// TwinCAT 3 PLC project PLC1
// ProgramVersion: 3.1.4026.15
// libraries:
//   Tc2_ModbusRTU, * (Beckhoff Automation GmbH)
//   Tc2_ModbusSrv, * (Beckhoff Automation GmbH)
//   Tc2_Standard, * (Beckhoff Automation GmbH)
//   Tc2_System, * (Beckhoff Automation GmbH)
// project tree:
//   GVLs/ FIO.TcGVL, GVL.TcGVL
//   / PlcTask.TcTTO
//   POUs/FactoryIO/ AssignInsOuts.TcPOU
//   POUs/FactoryIO/NOT USED/ FB_FactoryIO_ReadInputs_.TcPOU, FB_FactoryIO_WriteOutputs.TcPOU
//   POUs/ MAIN.TcPOU
//   POUs/SubRoutines/ F_Faults.TcPOU, C_Input_Conveyor.TcPOU, B_Machine_Center.TcPOU, E_Output_Conveyor.TcPOU, D_Stacker_Crane.TcPOU, A_System_Start.TcPOU
// real-time tasks:
//   TASK PlcTask: cycle T#10ms, priority 20, ADS port 350

CONFIGURATION PLC1
    RESOURCE PLC ON TwinCAT3
        TASK PlcTask(INTERVAL := T#10ms, PRIORITY := 20);
        PROGRAM MAIN WITH PlcTask : MAIN;
    END_RESOURCE
END_CONFIGURATION

// ---- GVLs/FIO.TcGVL
{attribute 'qualified_only'}
VAR_GLOBAL
	
//HMI
	



//Factory IO 
	//Inputs
		// MACH CNTR BUSY
			b_IN_0: BOOL;
		// MACH CNTR ERR
			b_IN_1: BOOL;
		// CONTAIN EMIT PE
			b_IN_2: BOOL;
		// BASE VISION SENS
			b_IN_3: BOOL;
		// INPUT CONV 1 PE
			b_IN_4: BOOL;
		// INPUT PICKUP PE
			b_IN_5: BOOL;
		// OUT DEP CONV PE
			b_IN_6: BOOL;
		// OUT CONV 1 PE
			b_IN_7: BOOL;
		// OUT CONV 2 PE
			b_IN_8: BOOL;
		// CRANE MOVE X
			b_IN_9: BOOL;
		// CRANE MOVE Z
			b_IN_10: BOOL;
		// CRANE LEFT LS
			b_IN_11: BOOL;
		// CRANE RIGHT LS
			b_IN_12: BOOL;
		// CRANE MID LS
			b_IN_13: BOOL;
		// UNUSED
			b_IN_14: BOOL;
		// UNUSED
			b_IN_15: BOOL;
		// UNUSED
			b_IN_64: BOOL;
	
	
		// Machining Center  Progress
			r_IN_0: WORD;
		//Light Array Emitter
			r_IN_1: WORD;
//Outputs
		// RAW MAT EMIT
			b_OUT_0: BOOL;
		// MACH LIDS
			b_OUT_1: BOOL;
		// CONTAIN CONV EMIT
			b_OUT_2: BOOL;
		// CONTAIN CONV MS
			b_OUT_3: BOOL := FALSE;
		// CONV PICK MS
			b_OUT_4: BOOL;
		// OUT DEP CONV MS
			b_OUT_5: BOOL;
		// OUT CONV 1 MS
			b_OUT_6: BOOL;
		// OUT CONV 2 MS
			b_OUT_7: BOOL;
		// OUT CONV REMOVE
			b_OUT_8: BOOL;
		// CRANE LIFT
			b_OUT_9: BOOL;
		// CRANE LEFT
			b_OUT_10: BOOL;
		// CRANE RIGHT
			b_OUT_11: BOOL;
		// INPUT CONV 1 MS
			b_OUT_12: BOOL;
		// CNC MACH RESET
			b_OUT_13: BOOL;
		// UNUSED
			b_OUT_14: BOOL;
		// UNUSED
			b_OUT_15: BOOL;
		// UNUSED
			b_OUT_16: BOOL;
		
		
		//Stacker Crane Target Position
			r_out_0: WORD;

END_VAR

// ---- GVLs/GVL.TcGVL
{attribute 'qualified_only'}
VAR_GLOBAL
	bSystemStart : BOOL := FALSE; 			//HMI Start
    bAutoMode : BOOL := FALSE;				//HMI Auto
    bCNCOn : BOOL := FALSE;					//HMI CNC ON
    bRetrieveCMD : BOOL := FALSE;			//HMI Retrieve command
    bReset : BOOL := FALSE;					//HMI Reset

    iProductID : INT := 4000;				//Current Product ID
    arrStoredIDs : ARRAY[1..15] OF INT := [0];		//Array of stored products
    arrExitIDs : ARRAY[1..15] OF INT:= [0];		//Array of exited products
    iStorageCount : INT := 0;				//num of stored items
    iExitCount : INT := 0;					//num of retrieved items

    bFaultDetected : BOOL := FALSE;			//global fault indicator
    sFaultMessage : STRING := '';			//global fault message
	
	// Indicates System is in run state
	SystemRun: BOOL := FALSE;
	// Box ID of queued Container
	QueuedBoxID: INT := 0;
	// Box Waiting for crane
	ContainerWaitingInput: BOOL := FALSE;
	
	ContainerWaitingOutput : BOOL := FALSE;
	
	//Warehouse has reached 15 box capacity
	WarehouseFull : BOOL := FALSE;
	
	//If crane is in input mode
	InputtingBoxes : BOOL := TRUE;
	//If crane is in output mode
	OutputtingBoxes : BOOL := FALSE;
	//Commanded location of crane
	CommandedLocation : INT :=1;
END_VAR

// ---- POUs/MAIN.TcPOU
PROGRAM MAIN
VAR
END_VAR

AssignInsOuts();


A_System_Start();
IF gvl.bSystemStart THEN
	IF GVL.SystemRun THEN
		B_Machine_Center();
		C_Input_Conveyor();
		D_Stacker_Crane();
		E_Output_Conveyor();
	END_IF
    F_Faults();
END_IF

END_PROGRAM

// ---- POUs/FactoryIO/AssignInsOuts.TcPOU
PROGRAM AssignInsOuts
VAR
	//Factory IO
	FactoryIO_Ins : ARRAY [0..15] OF BYTE;
	FactoryIO_RegIns : ARRAY [0..7] OF WORD;
	FactoryIO_Outs : ARRAY [0..15] OF BYTE;
	FactoryIO_RegOuts : ARRAY [0..7] OF WORD;
	
	//FIO Function Blocks
	FactoryIO_ReadInsFB : FB_MBReadInputs;
	FactoryIO_WriteOutsFB : FB_MBWriteCoils;
	FactoryIO_ReadRegsFB : FB_MBReadInputRegs;
	FactoryIO_WriteRegsFB : FB_MBWriteRegs;
	
END_VAR

//Reads Inputs and Writes Outputs to FactoryIO


FactoryIO_ReadInsFB(
	sIPAddr:= '127.0.0.1' , 
	nTCPPort:= 505, 
	nUnitID:= 1, 
	nQuantity:= 16, 
	nMBAddr:= 0, 
	cbLength:= SIZEOF(AssignInsOuts.FactoryIO_Ins), 
	pDestAddr:= ADR(AssignInsOuts.FactoryIO_Ins), 
	bExecute:= TRUE, 
	tTimeout:= T#1S, 
	bBusy=> , 
	bError=> , 
	nErrId=> , 
	cbRead=> );
FactoryIO_ReadInsFB(bExecute:=FALSE);


FactoryIO_ReadRegsFB(
	sIPAddr:= '127.0.0.1', 
	nTCPPort:= 505, 
	nUnitID:= 1, 
	nQuantity:= 8, 
	nMBAddr:= 0, 
	cbLength:=  SIZEOF(AssignInsOuts.FactoryIO_RegIns), 
	pDestAddr:= ADR(AssignInsOuts.FactoryIO_RegIns), 
	bExecute:= TRUE, 
	tTimeout:= T#1S, 
	bBusy=> , 
	bError=> , 
	nErrId=> , 
	cbRead=> );
FactoryIO_ReadRegsFB(bExecute := FALSE);



FactoryIO_WriteOutsFB(
	sIPAddr:= '127.0.0.1', 
	nTCPPort:= 505, 
	nUnitID:= 1, 
	nQuantity:= 16, 
	nMBAddr:= 0, 
	cbLength:= SIZEOF(AssignInsOuts.FactoryIO_Outs), 
	pSrcAddr:= ADR(AssignInsOuts.FactoryIO_Outs), 
	bExecute:= TRUE, 
	tTimeout:= T#1S, 
	bBusy=> , 
	bError=> , 
	nErrId=> );
FactoryIO_WriteOutsFB(bExecute:=FALSE);



FactoryIO_WriteRegsFB(
	sIPAddr:= '127.0.0.1', 
	nTCPPort:= 505, 
	nUnitID:= 1, 
	nQuantity:= 8, 
	nMBAddr:= 0, 
	cbLength:= SIZEOF(AssignInsOuts.FactoryIO_regOuts), 
	pSrcAddr:= ADR(AssignInsOuts.FactoryIO_regOuts), 
	bExecute:= TRUE, 
	tTimeout:= T#1S, 
	bBusy=> , 
	bError=> , 
	nErrId=> );
FactoryIO_WriteRegsFB(bExecute := FALSE);
	




//Link Inputs from FactoryIO
FIO.b_IN_0 :=  FactoryIO_Ins [0].0;
FIO.b_IN_1 :=  FactoryIO_Ins [0].1;
FIO.b_IN_2 :=  FactoryIO_Ins [0].2;
FIO.b_IN_3 :=  FactoryIO_Ins [0].3;
FIO.b_IN_4 :=  FactoryIO_Ins [0].4;
FIO.b_IN_5 :=  FactoryIO_Ins [0].5;
FIO.b_IN_6 :=  FactoryIO_Ins [0].6;
FIO.b_IN_7 :=  FactoryIO_Ins [0].7;
FIO.b_IN_8 :=  FactoryIO_Ins [1].0;
FIO.b_IN_9 :=  FactoryIO_Ins [1].1;
FIO.b_IN_10 :=  FactoryIO_Ins [1].2;
FIO.b_IN_11 :=  FactoryIO_Ins [1].3;
FIO.b_IN_12 :=  FactoryIO_Ins [1].4;
FIO.b_IN_13 :=  FactoryIO_Ins [1].5;
FIO.b_IN_14 :=  FactoryIO_Ins [1].6;
FIO.b_IN_15 :=  FactoryIO_Ins [1].6;

FIO.r_IN_0 := FactoryIO_RegIns [0];
FIO.r_IN_1 := FactoryIO_RegIns [1];


//Link Outputs to FactoryIO
FactoryIO_Outs [0].0 := FIO.b_OUT_0;
FactoryIO_Outs [0].1 := FIO.b_OUT_1;
FactoryIO_Outs [0].2 := FIO.b_OUT_2;
FactoryIO_Outs [0].3 := FIO.b_OUT_3;
FactoryIO_Outs [0].4 := FIO.b_OUT_4;
FactoryIO_Outs [0].5 := FIO.b_OUT_5;
FactoryIO_Outs [0].6 := FIO.b_OUT_6;
FactoryIO_Outs [0].7 := FIO.b_OUT_7;
FactoryIO_Outs [1].0 := FIO.b_OUT_8;
FactoryIO_Outs [1].1 := FIO.b_OUT_9;
FactoryIO_Outs [1].2 := FIO.b_OUT_10;
FactoryIO_Outs [1].3 := FIO.b_OUT_11;
FactoryIO_Outs [1].4 := FIO.b_OUT_12;
FactoryIO_Outs [1].5 := FIO.b_OUT_13;

FactoryIO_RegOuts[0] := FIO.r_out_0;

END_PROGRAM

// ---- POUs/SubRoutines/A_System_Start.TcPOU
PROGRAM A_System_Start
VAR

	INITIALIZED: BOOL;
	i: INT;
END_VAR




IF GVL.bSystemStart AND NOT GVL.SystemRun AND NOT INITIALIZED THEN	
	INITIALIZED := TRUE;
	GVL.SystemRun := TRUE;
	FIO.b_OUT_2 := TRUE;//Starts Emitter
	FIO.b_OUT_3 := FALSE;// Stops conveyor 1
	FIO.b_OUT_12 := FALSE;// Stops Conveyor 2
	FIO.b_OUT_4 := FALSE;// Stops Conveyor 3
	gvl.iProductID := 4000;
	GVL.QueuedBoxID := 0;
	
	FOR i := 0 TO 15 DO
		GVL.arrStoredIDs[i] := 0;
		GVL.arrExitIDs[i] := 0;
	END_FOR;
	gvl.CommandedLocation := 1;
	gvl.InputtingBoxes := TRUE;
	GVL.OutputtingBoxes := FALSE;
END_IF

GVL.SystemRun := GVL.bSystemStart;

IF GVL.bReset THEN
	GVL.SystemRun := FALSE;
	INITIALIZED := FALSE;
END_IF

END_PROGRAM

// ---- POUs/SubRoutines/B_Machine_Center.TcPOU
PROGRAM B_Machine_Center
VAR

END_VAR

FIO.b_OUT_1 := FALSE;
FIO.b_OUT_0 := FALSE; //Sets raw emitter to default off
IF (NOT FIO.b_IN_0) AND FIO.b_IN_2  THEN
	FIO.b_OUT_0 := TRUE;
	FIO.b_OUT_1 := TRUE;
	
END_IF

END_PROGRAM

// ---- POUs/SubRoutines/C_Input_Conveyor.TcPOU
PROGRAM C_Input_Conveyor
VAR


END_VAR


// When no containers queued for crane.
IF NOT GVL.ContainerWaitingInput THEN 
	//If there is a full container, move it along the conveyor
	IF FIO.b_IN_2 AND FIO.b_IN_3 THEN
		FIO.b_OUT_2 := FALSE;//Stops Emitter
		FIO.b_OUT_3 := TRUE;// Starts Conveyor 1
		FIO.b_OUT_12 := TRUE;// Starts Conveyor 2
	END_IF
	
	//If the conveyor reaches the first sensor, it stops the first section of the conveyor, starts the third, and emits a new empty container
	IF  FIO.b_IN_4 THEN
		FIO.b_OUT_2 := TRUE; // Emit new container
		FIO.b_OUT_3 := FALSE;// Stops conveyor 1
		FIO.b_OUT_12 := TRUE;// Starts Conveyor 2
		FIO.b_OUT_4 := TRUE;// Starts Conveyor 3
	END_IF
	//If the crane has a container in its loading queue, it stops the conveyor until it is picked up.
	IF  FIO.b_IN_5 THEN
		FIO.b_OUT_2 := FALSE;//Stops emitter
		//GVL.QueuedBoxID := GVL.iProductID;
		//GVL.iProductID := GVL.iProductID +1;
		GVL.ContainerWaitingInput := TRUE;//Sets box waiting to true
		FIO.b_OUT_12 := FALSE;	// stops conveyor 2
		FIO.b_OUT_4 := FALSE;	//stops conveyor 3
	END_IF
END_IF

// If one container is queued for crane
IF GVL.ContainerWaitingInput THEN 
	//If there is a full container, move it along the conveyor
	IF FIO.b_IN_2 AND FIO.b_IN_3 THEN
		FIO.b_OUT_3 := TRUE;// Starts Conveyor 1
		FIO.b_OUT_12 := TRUE;// Starts Conveyor 2
	END_IF
	
	//If the conveyor reaches the first sensor, it stops both sections of the conveyor
	IF  FIO.b_IN_4 THEN
		FIO.b_OUT_3 := FALSE;// Stops conveyor 1
		FIO.b_OUT_12 := FALSE;// Stops Conveyor 2
	END_IF
	
	//If the crane has a container in its loading queue, it stops the conveyor until it is picked up.
	IF  NOT FIO.b_IN_5 THEN
		GVL.ContainerWaitingInput := FALSE;//Sets container waiting to false. Switches to first statement
	END_IF
END_IF

END_PROGRAM

// ---- POUs/SubRoutines/D_Stacker_Crane.TcPOU
PROGRAM D_Stacker_Crane
VAR

	// Current Crane position state
	CranePosition: INT := 0;
	timer : TON;

END_VAR




IF gvl.InputtingBoxes AND (NOT GVL.OutputtingBoxes) THEN
	CASE CranePosition OF
	0://Waiting for command
		FIO.r_out_0:= 99; 		// Crane Position
		FIO.b_OUT_9 := FALSE; 	// Crane Lift
		FIO.b_OUT_10 := FALSE;	//Crane Left (DROPOFF)
		FIO.b_OUT_11 := FALSE;	//Crane Right (Receive)
		timer(IN:= TRUE, PT:= T#500MS, Q=> , ET=> );
		IF GVL.ContainerWaitingInput AND timer.q THEN
			CranePosition := 1;
			timer(IN := FALSE);
		END_IF
	1://Default Position lowered
		FIO.r_out_0:= 99; 		// Crane Position
		FIO.b_OUT_9 := FALSE; 	// Crane Lift
		FIO.b_OUT_10 := FALSE;	//Crane Left (DROPOFF)
		FIO.b_OUT_11 := FALSE;	//Crane Right (Receive)
		timer(IN:= TRUE, PT:= T#500MS, Q=> , ET=> );
		IF (NOT (FIO.b_IN_9 OR FIO.b_IN_10)) AND FIO.b_IN_13 AND timer.q THEN
			CranePosition := 10;
			timer(IN := FALSE);
		END_IF
	10://Pickup lowered
		FIO.r_out_0:= 99; 		// Crane Position
		FIO.b_OUT_9 := FALSE; 	// Crane Lift
		FIO.b_OUT_10 := FALSE;	//Crane Left (DROPOFF)
		FIO.b_OUT_11 := TRUE;	//Crane Right (Receive)
		timer(IN:= TRUE, PT:= T#500MS, Q=> , ET=> );
		IF (NOT (FIO.b_IN_9 OR FIO.b_IN_10)) AND FIO.b_IN_12 AND timer.q THEN
			CranePosition := 20;
			timer(IN := FALSE);
		END_IF
	20://Pickup raised
		FIO.r_out_0:= 99; 		// Crane Position
		FIO.b_OUT_9 := TRUE; 	// Crane Lift
		FIO.b_OUT_10 := FALSE;	//Crane Left (DROPOFF)
		FIO.b_OUT_11 := TRUE;	//Crane Right (Receive)
		timer(IN:= TRUE, PT:= T#500MS, Q=> , ET=> );
		IF timer.Q  THEN
			CranePosition := 30;
			timer(IN := FALSE);
		END_IF
	30://DefaultPosition raised
		FIO.r_out_0:= 99; 		// Crane Position
		FIO.b_OUT_9 := TRUE; 	// Crane Lift
		FIO.b_OUT_10 := FALSE;	//Crane Left (DROPOFF)
		FIO.b_OUT_11 := FALSE;	//Crane Right (Receive)
		IF (NOT (FIO.b_IN_9 OR FIO.b_IN_10)) AND FIO.b_IN_13  THEN
			CranePosition := 40;
		END_IF
	40://Commanded Location queue lowered
		FIO.r_out_0:= TO_WORD(gvl.CommandedLocation); 		// Crane Position
		FIO.b_OUT_9 := FALSE; 	// Crane Lift
		FIO.b_OUT_10 := FALSE;	//Crane Left (DROPOFF)
		FIO.b_OUT_11 := FALSE;	//Crane Right (Receive)
		timer(IN:= TRUE, PT:= T#500MS, Q=> , ET=> );
		IF (NOT FIO.b_IN_9) AND (NOT FIO.b_IN_10) AND FIO.b_IN_13 AND timer.q THEN
			CranePosition := 50;
			timer(IN := FALSE);
		END_IF
	50://Commanded Location queue raised
		FIO.r_out_0:= TO_WORD(gvl.CommandedLocation); 		// Crane Position
		FIO.b_OUT_9 := TRUE; 	// Crane Lift
		FIO.b_OUT_10 := FALSE;	//Crane Left (DROPOFF)
		FIO.b_OUT_11 := FALSE;	//Crane Right (Receive)
		timer(IN:= TRUE, PT:= T#500MS, Q=> , ET=> );
		IF (NOT (FIO.b_IN_9 OR FIO.b_IN_10)) AND FIO.b_IN_13  AND Timer.q THEN
			CranePosition := 60;
			timer(IN := FALSE);
		END_IF
	60://Commanded Location raised
		FIO.r_out_0:= TO_WORD(gvl.CommandedLocation); 		// Crane Position
		FIO.b_OUT_9 := TRUE; 	// Crane Lift
		FIO.b_OUT_10 := TRUE;	//Crane Left (DROPOFF)
		FIO.b_OUT_11 := FALSE;	//Crane Right (Receive)
		timer(IN:= TRUE, PT:= T#500MS, Q=> , ET=> );
		IF (NOT (FIO.b_IN_9 OR FIO.b_IN_10)) AND FIO.b_IN_11 AND Timer.q THEN
			CranePosition := 70;
			timer(IN := FALSE);
		END_IF
	70://Commanded Location lowered
		FIO.r_out_0:= TO_WORD(gvl.CommandedLocation); 		// Crane Position
		FIO.b_OUT_9 := FALSE; 	// Crane Lift
		FIO.b_OUT_10 := TRUE;	//Crane Left (DROPOFF)
		FIO.b_OUT_11 := FALSE;	//Crane Right (Receive)
		timer(IN:= TRUE, PT:= T#500MS, Q=> , ET=> );
		GVL.arrStoredIDs[GVL.CommandedLocation] := GVL.iProductID; 
		IF (NOT (FIO.b_IN_9 OR FIO.b_IN_10)) AND FIO.b_IN_11 AND timer.q THEN
			CranePosition := 80;
			timer(IN := FALSE);
			GVL.arrStoredIDs[GVL.CommandedLocation] := GVL.iProductID; 
			GVL.iProductID := GVL.iProductID +1;
		END_IF
	80://Commanded Location queue lowered
		FIO.r_out_0:= TO_WORD(gvl.CommandedLocation); 		// Crane Position
		FIO.b_OUT_9 := FALSE; 	// Crane Lift
		FIO.b_OUT_10 := FALSE;	//Crane Left (DROPOFF)
		FIO.b_OUT_11 := FALSE;	//Crane Right (Receive)
		timer(IN:= TRUE, PT:= T#500MS, Q=> , ET=> );
		IF (NOT (FIO.b_IN_9 OR FIO.b_IN_10)) AND FIO.b_IN_13 AND timer.q THEN
			CranePosition := 0;
			timer(IN := FALSE);	
			IF gvl.CommandedLocation < 15 THEN
				gvl.CommandedLocation := gvl.CommandedLocation +1;
			ELSIF gvl.CommandedLocation = 15 THEN
				gvl.WarehouseFull := TRUE;
				gvl.CommandedLocation := 1;
				GVL.InputtingBoxes := FALSE;
				GVL.OutputtingBoxes := TRUE;
			END_IF
		END_IF
END_CASE
END_IF

IF gvl.OutputtingBoxes AND (NOT GVL.InputtingBoxes) THEN
	CASE CranePosition OF
	0://Default Position lowered
		FIO.r_out_0:= 99; 		// Crane Position
		FIO.b_OUT_9 := FALSE; 	// Crane Lift
		FIO.b_OUT_10 := FALSE;	//Crane Left (DROPOFF)
		FIO.b_OUT_11 := FALSE;	//Crane Right (Receive)
		timer(IN:= TRUE, PT:= T#500MS, Q=> , ET=> );
		IF (NOT (FIO.b_IN_9 OR FIO.b_IN_10)) AND FIO.b_IN_13 AND timer.q THEN
			CranePosition := 10;
			timer(IN := FALSE);
		END_IF
	
	10://Commanded Location queue lowered
		FIO.r_out_0:= TO_WORD(gvl.CommandedLocation); 		// Crane Position
		FIO.b_OUT_9 := FALSE; 	// Crane Lift
		FIO.b_OUT_10 := FALSE;	//Crane Left (DROPOFF)
		FIO.b_OUT_11 := FALSE;	//Crane Right (Receive)
		timer(IN:= TRUE, PT:= T#500MS, Q=> , ET=> );
		IF (NOT FIO.b_IN_9) AND (NOT FIO.b_IN_10) AND FIO.b_IN_13 AND timer.q THEN
			CranePosition := 20;
			timer(IN := FALSE);
		END_IF
	20://Commanded Location lowered
		FIO.r_out_0:= TO_WORD(gvl.CommandedLocation); 		// Crane Position
		FIO.b_OUT_9 := FALSE; 	// Crane Lift
		FIO.b_OUT_10 := TRUE;	//Crane Left (DROPOFF)
		FIO.b_OUT_11 := FALSE;	//Crane Right (Receive)
		timer(IN:= TRUE, PT:= T#500MS, Q=> , ET=> );
		IF (NOT (FIO.b_IN_9 OR FIO.b_IN_10)) AND FIO.b_IN_11 AND timer.q THEN
			CranePosition := 30;
			timer(IN := FALSE);
		END_IF
	30://Commanded Location raised
		FIO.r_out_0:= TO_WORD(gvl.CommandedLocation); 		// Crane Position
		FIO.b_OUT_9 := TRUE; 	// Crane Lift
		FIO.b_OUT_10 := TRUE;	//Crane Left (DROPOFF)
		FIO.b_OUT_11 := FALSE;	//Crane Right (Receive)
		timer(IN:= TRUE, PT:= T#500MS, Q=> , ET=> );
		IF (NOT (FIO.b_IN_9 OR FIO.b_IN_10)) AND FIO.b_IN_11 AND Timer.q THEN
			CranePosition := 40;
			timer(IN := FALSE);
		END_IF
	40://Commanded Location queue raised
		FIO.r_out_0:= TO_WORD(gvl.CommandedLocation); 		// Crane Position
		FIO.b_OUT_9 := TRUE; 	// Crane Lift
		FIO.b_OUT_10 := FALSE;	//Crane Left (DROPOFF)
		FIO.b_OUT_11 := FALSE;	//Crane Right (Receive)
		timer(IN:= TRUE, PT:= T#500MS, Q=> , ET=> );
		IF (NOT (FIO.b_IN_9 OR FIO.b_IN_10)) AND FIO.b_IN_13  AND Timer.q THEN
			CranePosition := 50;
			timer(IN := FALSE);
		END_IF
	50://Commanded Location queue lowered
		FIO.r_out_0:= TO_WORD(gvl.CommandedLocation); 		// Crane Position
		FIO.b_OUT_9 := FALSE; 	// Crane Lift
		FIO.b_OUT_10 := FALSE;	//Crane Left (DROPOFF)
		FIO.b_OUT_11 := FALSE;	//Crane Right (Receive)
		timer(IN:= TRUE, PT:= T#500MS, Q=> , ET=> );
		IF (NOT (FIO.b_IN_9 OR FIO.b_IN_10)) AND FIO.b_IN_13 AND timer.q THEN
			CranePosition := 60;
			timer(IN := FALSE);
		END_IF
	60://Default Position Raised
		FIO.r_out_0:= 99; 		// Crane Position
		FIO.b_OUT_9 := TRUE; 	// Crane Lift
		FIO.b_OUT_10 := FALSE;	//Crane Left (DROPOFF)
		FIO.b_OUT_11 := FALSE;	//Crane Right (Receive)
		timer(IN:= TRUE, PT:= T#500MS, Q=> , ET=> );
		IF (NOT (FIO.b_IN_9 OR FIO.b_IN_10)) AND FIO.b_IN_13 AND timer.q AND NOT GVL.ContainerWaitingOutput THEN
			CranePosition := 70;
			timer(IN := FALSE);
		END_IF
	70://Deposit raised
		FIO.r_out_0:= 99; 		// Crane Position
		FIO.b_OUT_9 := TRUE; 	// Crane Lift
		FIO.b_OUT_10 := TRUE;	//Crane Left (DROPOFF)
		FIO.b_OUT_11 := FALSE;	//Crane Right (Receive)
		timer(IN:= TRUE, PT:= T#500MS, Q=> , ET=> );
		IF timer.Q  THEN
			CranePosition := 80;
			timer(IN := FALSE);
		END_IF	
	80://Deposit lowered
		FIO.r_out_0:= 99; 		// Crane Position
		FIO.b_OUT_9 := FALSE; 	// Crane Lift
		FIO.b_OUT_10 := TRUE;	//Crane Left (DROPOFF)
		FIO.b_OUT_11 := FALSE;	//Crane Right (Receive)
		timer(IN:= TRUE, PT:= T#500MS, Q=> , ET=> );
		IF timer.Q  THEN
			CranePosition := 90;
			timer(IN := FALSE);
			GVL.arrExitIDs[GVL.CommandedLocation] := GVL.arrStoredIDs[GVL.CommandedLocation]; 
		END_IF
	90://Default Position lowered
		FIO.r_out_0:= 99; 		// Crane Position
		FIO.b_OUT_9 := FALSE; 	// Crane Lift
		FIO.b_OUT_10 := FALSE;	//Crane Left (DROPOFF)
		FIO.b_OUT_11 := FALSE;	//Crane Right (Receive)
		timer(IN:= TRUE, PT:= T#500MS, Q=> , ET=> );
		IF (NOT (FIO.b_IN_9 OR FIO.b_IN_10)) AND FIO.b_IN_13 AND timer.q THEN
			CranePosition := 0;
			timer(IN := FALSE);	
			IF gvl.CommandedLocation < 15 THEN
				gvl.CommandedLocation := gvl.CommandedLocation +1;
			ELSIF gvl.CommandedLocation = 15 THEN
				gvl.WarehouseFull := FALSE;
				gvl.CommandedLocation := 1;
				GVL.InputtingBoxes := TRUE;
				GVL.OutputtingBoxes := FALSE;
			END_IF
		END_IF
END_CASE
END_IF

END_PROGRAM

// ---- POUs/SubRoutines/E_Output_Conveyor.TcPOU
PROGRAM E_Output_Conveyor
VAR

WaitTimer : TON;

END_VAR




GVL.ContainerWaitingOutput := FIO.b_IN_6;


IF GVL.ContainerWaitingOutput AND NOT FIO.b_IN_7  THEN
	FIO.b_OUT_5 := TRUE;
	FIO.b_OUT_6 := TRUE;
END_IF

IF FIO.b_IN_7 AND NOT FIO.b_IN_8 THEN
	FIO.b_OUT_5 := FALSE;
	FIO.b_OUT_6 := TRUE;
	FIO.b_OUT_7 := TRUE;
END_IF
IF FIO.b_IN_7 AND  FIO.b_IN_8 THEN
	FIO.b_OUT_5 := FALSE;
	FIO.b_OUT_6 := FALSE;
	FIO.b_OUT_7 := FALSE;
END_IF

IF FIO.b_IN_8 THEN
	IF NOT FIO.b_OUT_5 THEN
		FIO.b_OUT_6 := FALSE;
	END_IF
	FIO.b_OUT_7 := FALSE;
	WaitTimer(IN:= TRUE, PT:= T#10S, Q=> , ET=> );
ELSE
	WaitTimer(IN:= FALSE, PT:= T#10S, Q=> , ET=> );
END_IF
FIO.b_OUT_8 := WaitTimer.Q;

END_PROGRAM

// ---- POUs/SubRoutines/F_Faults.TcPOU
PROGRAM F_Faults
VAR

END_VAR

IF FIO.b_IN_1 AND GVL.bReset THEN 
	FIO.b_OUT_13 := TRUE;
ELSE
	FIO.b_OUT_13 := FALSE;
END_IF

END_PROGRAM

// ---- POUs/FactoryIO/NOT USED/FB_FactoryIO_ReadInputs_.TcPOU
FUNCTION_BLOCK FB_FactoryIO_ReadInputs_
VAR_INPUT
END_VAR
VAR_OUTPUT
END_VAR
VAR
	FactoryIO_ReadInsFB : FB_MBReadInputs;
	
END_VAR

FactoryIO_ReadInsFB(
	sIPAddr:= '127.0.0.1' , 
	nTCPPort:= 75, 
	nUnitID:= 1, 
	nQuantity:= 16, 
	nMBAddr:= 0, 
	cbLength:= SIZEOF(AssignInsOuts.FactoryIO_Ins), 
	pDestAddr:= ADR(AssignInsOuts.FactoryIO_Ins), 
	bExecute:= TRUE, 
	tTimeout:= T#1S, 
	bBusy=> , 
	bError=> , 
	nErrId=> , 
	cbRead=> );

FactoryIO_ReadInsFB(bExecute:=FALSE);

END_FUNCTION_BLOCK

// ---- POUs/FactoryIO/NOT USED/FB_FactoryIO_WriteOutputs.TcPOU
FUNCTION_BLOCK FB_FactoryIO_WriteOutputs
VAR_INPUT
END_VAR
VAR_OUTPUT
END_VAR
VAR
	FactoryIO_WriteOutsFB : FB_MBWriteCoils;
END_VAR

FactoryIO_WriteOutsFB(
	sIPAddr:= '127.0.0.1', 
	nTCPPort:= 75, 
	nUnitID:= 1, 
	nQuantity:= 16, 
	nMBAddr:= 0, 
	cbLength:= SIZEOF(AssignInsOuts.FactoryIO_Outs), 
	pSrcAddr:= ADR(AssignInsOuts.FactoryIO_Outs), 
	bExecute:= TRUE, 
	tTimeout:= T#1S, 
	bBusy=> , 
	bError=> , 
	nErrId=> );
	
	FactoryIO_WriteOutsFB(bExecute:=FALSE);

END_FUNCTION_BLOCK
